// TIA Portal V18 export
DATA_BLOCK "Working_Sequence_DB"   // DB8
VERSION : 0.1
// stored: AutoNumber true, InstanceOfName Working_Sequence, InstanceOfType FB
"Working_Sequence"
BEGIN
END_DATA_BLOCK
